PROGRAM Motion_Step
VAR
	Axis04_Torque_Controll: TON;
	Axis02_Wait_Pos_Moving_Delay: TON;
	Always_ON	:	BOOL	:=TRUE	;//상시 ON 
	Always_OFF	:	BOOL	:=FALSE	;//상시 OFF
	Axis04_Work_end_Delay: TON;
END_VAR
VAR // added by the converter: edge detectors and wires of the graphical bodies
    _rt1 : R_TRIG;
    _w1, _w2, _w3, _w4, _w5, _w6, _w7, _w8, _w9, _w10, _w11, _w12 : BOOL;
END_VAR

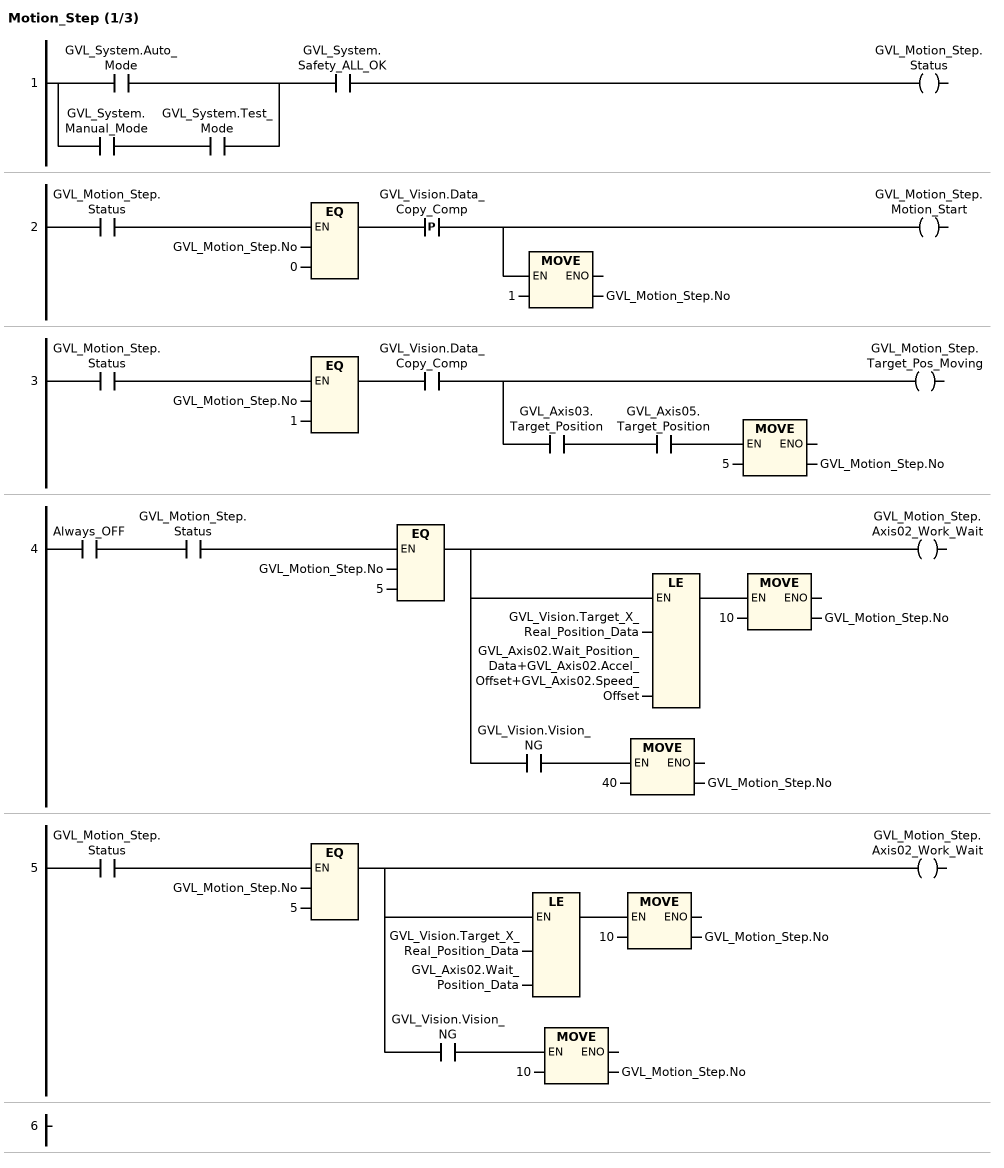
// NETWORK 1
GVL_Motion_Step.Status := (GVL_System.Auto_Mode OR GVL_System.Manual_Mode AND GVL_System.Test_Mode) AND GVL_System.Safety_ALL_OK;

// NETWORK 2
_rt1(CLK := GVL_Vision.Data_Copy_Comp);
_w1 := (GVL_Motion_Step.Status AND GVL_Motion_Step.No = 0) AND _rt1.Q;
GVL_Motion_Step.Motion_Start := _w1;
IF _w1 THEN GVL_Motion_Step.No := 1; END_IF

// NETWORK 3
_w2 := (GVL_Motion_Step.Status AND GVL_Motion_Step.No = 1) AND GVL_Vision.Data_Copy_Comp;
GVL_Motion_Step.Target_Pos_Moving := _w2;
IF _w2 AND GVL_Axis03.Target_Position AND GVL_Axis05.Target_Position THEN GVL_Motion_Step.No := 5; END_IF

// NETWORK 4
_w3 := Always_OFF AND GVL_Motion_Step.Status AND GVL_Motion_Step.No = 5;
GVL_Motion_Step.Axis02_Work_Wait := _w3;
IF _w3 AND GVL_Vision.Target_X_Real_Position_Data <= (GVL_Axis02.Wait_Position_Data+GVL_Axis02.Accel_Offset+GVL_Axis02.Speed_Offset) THEN
    GVL_Motion_Step.No := 10;
END_IF
IF _w3 AND GVL_Vision.Vision_NG THEN GVL_Motion_Step.No := 40; END_IF

// NETWORK 5
_w4 := GVL_Motion_Step.Status AND GVL_Motion_Step.No = 5;
GVL_Motion_Step.Axis02_Work_Wait := _w4;
IF _w4 AND GVL_Vision.Target_X_Real_Position_Data <= GVL_Axis02.Wait_Position_Data THEN
    GVL_Motion_Step.No := 10;
END_IF
IF _w4 AND GVL_Vision.Vision_NG THEN GVL_Motion_Step.No := 10; END_IF

// NETWORK 6

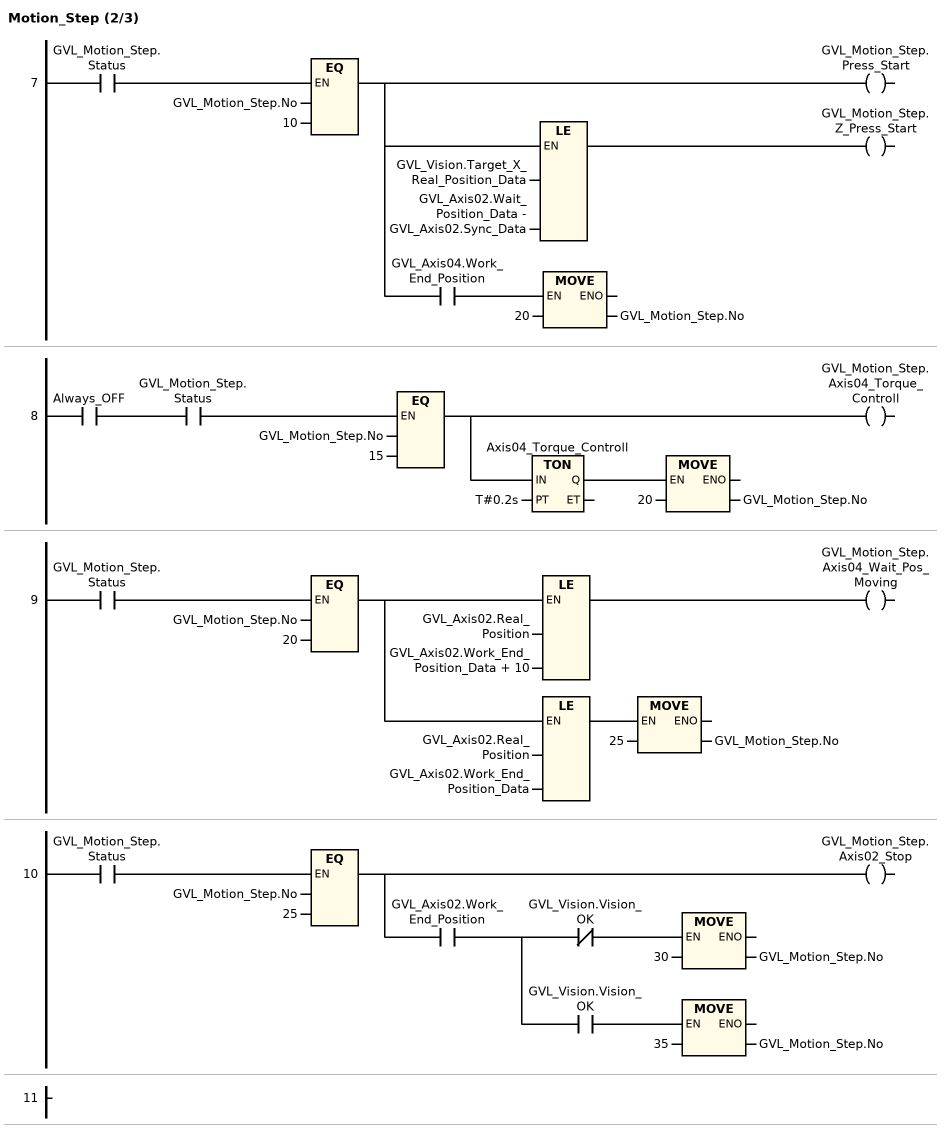
// NETWORK 7
_w5 := GVL_Motion_Step.Status AND GVL_Motion_Step.No = 10;
GVL_Motion_Step.Press_Start := _w5;
GVL_Motion_Step.Z_Press_Start := _w5 AND GVL_Vision.Target_X_Real_Position_Data <= (GVL_Axis02.Wait_Position_Data - GVL_Axis02.Sync_Data);
IF _w5 AND GVL_Axis04.Work_End_Position THEN GVL_Motion_Step.No := 20; END_IF

// NETWORK 8
_w6 := Always_OFF AND GVL_Motion_Step.Status AND GVL_Motion_Step.No = 15;
GVL_Motion_Step.Axis04_Torque_Controll := _w6;
Axis04_Torque_Controll(IN := _w6, PT := T#0.2s); // TON
IF Axis04_Torque_Controll.Q THEN GVL_Motion_Step.No := 20; END_IF

// NETWORK 9
_w7 := GVL_Motion_Step.Status AND GVL_Motion_Step.No = 20;
GVL_Motion_Step.Axis04_Wait_Pos_Moving := _w7 AND GVL_Axis02.Real_Position <= (GVL_Axis02.Work_End_Position_Data + 10);
IF _w7 AND GVL_Axis02.Real_Position <= GVL_Axis02.Work_End_Position_Data THEN GVL_Motion_Step.No := 25; END_IF

// NETWORK 10
_w8 := GVL_Motion_Step.Status AND GVL_Motion_Step.No = 25;
GVL_Motion_Step.Axis02_Stop := _w8;
_w9 := _w8 AND GVL_Axis02.Work_End_Position;
IF _w9 AND NOT GVL_Vision.Vision_OK THEN GVL_Motion_Step.No := 30; END_IF
IF _w9 AND GVL_Vision.Vision_OK THEN GVL_Motion_Step.No := 35; END_IF

// NETWORK 11

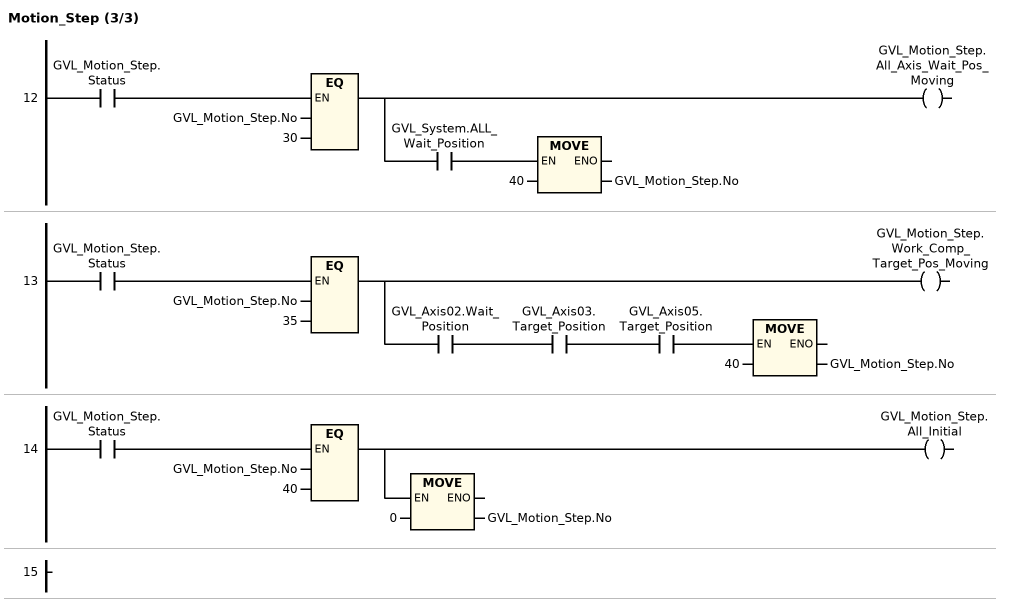
// NETWORK 12
_w10 := GVL_Motion_Step.Status AND GVL_Motion_Step.No = 30;
GVL_Motion_Step.All_Axis_Wait_Pos_Moving := _w10;
IF _w10 AND GVL_System.ALL_Wait_Position THEN GVL_Motion_Step.No := 40; END_IF

// NETWORK 13
_w11 := GVL_Motion_Step.Status AND GVL_Motion_Step.No = 35;
GVL_Motion_Step.Work_Comp_Target_Pos_Moving := _w11;
IF _w11 AND GVL_Axis02.Wait_Position AND GVL_Axis03.Target_Position AND GVL_Axis05.Target_Position THEN
    GVL_Motion_Step.No := 40;
END_IF

// NETWORK 14
_w12 := GVL_Motion_Step.Status AND GVL_Motion_Step.No = 40;
GVL_Motion_Step.All_Initial := _w12;
IF _w12 THEN GVL_Motion_Step.No := 0; END_IF

// NETWORK 15

END_PROGRAM

(* stored: Version 1.1.0.1, ProductVersion 3.1.4024.15
   POU Motion_Step: Id {2570e2ba-4534-4c79-8748-87544dc4a6b6}, SpecialFunc None *)
